Fanuc KAREL source: ka00066.KL

-- PROVISIONAL review KL for V1013-1; original PC SHA256 2a8dc6767c7712561b84ccdd5832e6e609f20b3991c0321afb42168b9ae0ad70
-- Incomplete behavior may be omitted. Consult companion uncertainty JSON. Do not deploy.
PROGRAM KA00066
%NOLOCKGROUP
-- UNRESOLVED_DECL SRC type=000102
-- UNRESOLVED_DECL DST type=000102
BEGIN
  -- UNRESOLVED_PC offsets 5-20; opcodes 2E,22,32,35
  -- UNRESOLVED_PC offsets 25-40; opcodes 49,4A
  -- UNRESOLVED_PC offsets 45-49; opcodes 7F
END KA00066
